// TIA Portal V19 export
TYPE "C402_VAR_IF_VKL_TYPIC"
   STRUCT
      STS_ROOD { ExternalAccessible := 'False'; ExternalVisible := 'False'; ExternalWritable := 'False'} : Bool;   // TRUE = Verkeerslicht actueel op rood
      STS_GEEL { ExternalAccessible := 'False'; ExternalVisible := 'False'; ExternalWritable := 'False'} : Bool;   // TRUE = Verkeerslicht actueel op geel (vast)
      STS_GROE { ExternalAccessible := 'False'; ExternalVisible := 'False'; ExternalWritable := 'False'} : Bool;   // TRUE = Verkeerslicht actueel op groen
      STS_KNIP { ExternalAccessible := 'False'; ExternalVisible := 'False'; ExternalWritable := 'False'} : Bool;   // TRUE = Verkeerslicht actueel op knipperen geel
      STS_AAN { ExternalAccessible := 'False'; ExternalVisible := 'False'; ExternalWritable := 'False'} : Bool;   // TRUE = Verkeerslicht wordt aangestuurd
      BMO_HAND { ExternalAccessible := 'False'; ExternalVisible := 'False'; ExternalWritable := 'False'} : Bool;   // TRUE = Verkeerslicht in hand geschakeld / FALSE = niet in hand
      EXT_AUT { ExternalAccessible := 'False'; ExternalVisible := 'False'; ExternalWritable := 'False'} : Bool;   // Externe (hoofd) beveiliging aangesproken
      EXT_HW { ExternalAccessible := 'False'; ExternalVisible := 'False'; ExternalWritable := 'False'} : Bool;   // Sturings hardware (PLC) in storing
      STO { ExternalAccessible := 'False'; ExternalVisible := 'False'; ExternalWritable := 'False'} : Struct   // Opsomming van alle signaleringen
         A001 : Bool;   // Beveiliging aangesproken
         AT01 : Bool;   // De rode lens is defect
         AT02 : Bool;   // De gele lens is defect
         AT03 : Bool;   // De groene lens is defect
         AT04 : Bool;   // De stand rood kan niet getoond worden
         AT05 : Bool;   // De stand geel kan niet getoond worden
         AT06 : Bool;   // De stand geel knipperen kan niet getoond worden
         AT07 : Bool;   // De stand groen kan niet getoond worden
      END_STRUCT;
   END_STRUCT;
END_TYPE
